// TIA Portal V18 export
// export: Created 2026-01-09T11:32:03.0527376Z, ExportSetting WithDefaults, DisplayName Totally Integrated Automation Portal, DisplayVersion V18 Update 5, DisplayName TIA Portal Openness, DisplayVersion V18 Update 5, DisplayName TIA Portal Teamcenter Gateway, DisplayVersion V18, DisplayName TIA Portal Version Control Interface, DisplayVersion V18, DisplayName SINAMICS Startdrive Advanced, DisplayVersion V18 SP2 Update 1, DisplayName SINAMICS Startdrive G110M, G120, G120C, G120D, G120P, G115D, DisplayVersion V18 SP2 Update 1, DisplayName SINAMICS Startdrive G130, G150, S120, S150, SINAMICS MV, S210, G220, S200, DisplayVersion V18 SP2 Update 1, DisplayName STEP 7 Professional, DisplayVersion V18 Update 5, DisplayName STEP 7 Safety, DisplayVersion V18, DisplayName WinCC Professional, DisplayVersion V18 Update 5
TagTable "C"
  Sys_ScanTime_CyclePrevious : Int  (PLC tag Sys.ScanTime.CyclePrevious, CPU S71500-2PN_TP700, 1 s)
  Sys_ScanTime_CycleMax : Int  (PLC tag Sys.ScanTime.CycleMax, CPU S71500-2PN_TP700, 1 s)
  Sys_ScanTime_CycleMin : Int  (PLC tag Sys.ScanTime.CycleMin, CPU S71500-2PN_TP700, 1 s)
  SysScanTimeCyclePrevious : Int  (PLC tag Sys.ScanTime.CyclePrevious, CPU S71500-2PN_TP700, 1 s)
  SysScanTimeCycleMax : Int  (PLC tag Sys.ScanTime.CycleMax, CPU S71500-2PN_TP700, 1 s)
  SysScanTimeCycleMin : Int  (PLC tag Sys.ScanTime.CycleMin, CPU S71500-2PN_TP700, 1 s)
